FUNCTION_BLOCK FB_PeerLinkedList EXTENDS FB_GenericLinkedList
VAR_INPUT
END_VAR
VAR_OUTPUT
END_VAR
VAR
END_VAR

METHOD M_AddPeerToHead : BOOL
VAR_INPUT
	pUnitToAdd : POINTER TO ST_LinkedListUnit;
	pPeerToAdd : POINTER TO ST_PeerAccount;
END_VAR
pUnitToAdd^.pVoid := pPeerToAdd;
SUPER^.M_AddToHead(pUnitToAdd);
END_METHOD

METHOD M_AddPeerToTail : BOOL
VAR_INPUT
	pUnitToAdd : POINTER TO ST_LinkedListUnit;
	pPeerToAdd : POINTER TO ST_PeerAccount;
END_VAR
pUnitToAdd^.pVoid := pPeerToAdd;
SUPER^.M_AddToTail(pUnitToAdd);
END_METHOD

METHOD M_GetHeadPeer : POINTER TO ST_PeerAccount
VAR_INPUT
END_VAR
VAR
	stUnit : POINTER TO ST_LinkedListUnit;
END_VAR
stUnit := SUPER^.M_GetHead();

IF stUnit = NULL THEN
	RETURN;
END_IF

M_GetHeadPeer := stUnit^.pVoid;
END_METHOD

METHOD M_GetNextPeer : POINTER TO ST_PeerAccount
VAR_INPUT
END_VAR
VAR
	stUnit : POINTER TO ST_LinkedListUnit;
END_VAR
stUnit := SUPER^.M_GetNext();

IF stUnit = NULL THEN
	RETURN;
END_IF

M_GetNextPeer := stUnit^.pVoid;
END_METHOD

METHOD M_GetTailPeer : POINTER TO ST_PeerAccount
VAR_INPUT
END_VAR
VAR
	stUnit : POINTER TO ST_LinkedListUnit;
END_VAR
stUnit := SUPER^.M_GetTail();

IF stUnit = NULL THEN
	RETURN;
END_IF

M_GetTailPeer := stUnit^.pVoid;
END_METHOD

END_FUNCTION_BLOCK

(* stored: Version 1.1.0.1, ProductVersion 3.1.4022.12
   POU FB_PeerLinkedList: Id {0929a248-657a-448c-9f2b-b51e90583290}, SpecialFunc None
   Method M_AddPeerToHead: Id {464f18b8-6c04-40f4-b288-175de2d0862d}
   Method M_AddPeerToTail: Id {3b77f470-7022-4971-b4ab-b206c5e3425d}
   Method M_GetHeadPeer: Id {d853f2c3-86cc-49ee-8bf7-ff0d989c9260}
   Method M_GetNextPeer: Id {636eccf5-2527-4f0a-8ddc-080149e32a15}
   Method M_GetTailPeer: Id {032d1d0b-1a07-4543-8e00-a69399b55fa1} *)
